// TwinCAT 3 PLC project FMStrings
// Title: FM Strings
// Company: FrameworkMonorepo
// ProjectVersion: 0.0.1
// ProgramVersion: 3.1.4024.0
// libraries:
//   FM Types, * (FrameworkMonorepo)
//   Tc2_Standard, * (Beckhoff Automation GmbH)
//   Tc2_System, * (Beckhoff Automation GmbH)
//   Tc2_Utilities, * (Beckhoff Automation GmbH)
//   Tc3_Module, * (Beckhoff Automation GmbH)
//   Base Interfaces,newest,System
// project tree:
//   Build/ BuildStringInline.TcPOU, StringBuilderExtBuffer.TcPOU, StringBuilder255.TcPOU, StringBuilderInfinite.TcPOU
//   Convert/ AnyToString.TcPOU, AnyTypeToString.TcPOU, StringToAny.TcPOU, StringToAnyType.TcPOU
//   Manipulate/ AddLeadingZeros.TcPOU, GetStringBetween.TcPOU, RemoveStringFromEnd.TcPOU, ReplaceAllAny.TcPOU, ReplaceAll.TcPOU, ReplaceAllAnyType.TcPOU, ReplaceString.TcPOU, SubString.TcPOU
//   Utf8/ Utf8String.TcDUT
//   Validate/ StringBeginsWithAny.TcPOU, StringBeginsWith.TcPOU, StringEndsWithAny.TcPOU, StringEndsWith.TcPOU
//   Version/ Global_Version.TcGVL
// (motion and I/O tree: see PLC project fmtypes)
// real-time tasks:
//   TASK BindingTestTask: cycle T#1ms, priority 20, ADS port 350
//   TASK PlcTask: cycle T#1ms, priority 21, ADS port 351
//   TASK PlcTask1: cycle T#1ms, priority 22, ADS port 352
//   TASK PlcTask2: cycle T#1ms, priority 23, ADS port 353
//   TASK MathTestTask: cycle T#1ms, priority 24, ADS port 354
//   TASK TimesTestsTask: cycle T#1ms, priority 25, ADS port 355

// ---- Utf8/Utf8String.TcDUT
{attribute 'TcEncoding':='UTF-8'}
TYPE Utf8String : T_MaxString; END_TYPE

// ---- Version/Global_Version.TcGVL
{attribute 'TcGenerated'}
{attribute 'no-analysis'}
{attribute 'linkalways'}
// This function has been automatically generated from the project information.
VAR_GLOBAL CONSTANT
	{attribute 'const_non_replaced'}
	stLibVersion_FM_Strings : ST_LibVersion := (iMajor := 0, iMinor := 0, iBuild := 1, iRevision := 0, nFlags := 0, sVersion := '0.0.1');
END_VAR

// ---- Build/BuildStringInline.TcPOU
FUNCTION BuildStringInline : REFERENCE TO StringBuilder255
VAR_INPUT
	value : T_MaxString;
END_VAR
VAR_STAT
	builder : StringBuilder255;
END_VAR

builder.Clear();

builder.Append(value);

BuildStringInline REF= builder;

END_FUNCTION

// ---- Build/StringBuilder255.TcPOU
FUNCTION_BLOCK StringBuilder255
VAR
	_Value : T_MaxString;
END_VAR

METHOD Append : REFERENCE TO StringBuilder255
VAR_INPUT
	value : T_MaxString;
END_VAR
Append REF= THIS^;

_Value := CONCAT(_Value, value);
END_METHOD

METHOD Clear : REFERENCE TO StringBuilder255
Clear REF= THIS^;

_Value := '';
END_METHOD

METHOD GetString : T_MaxString
GetString := _Value;
END_METHOD

PROPERTY IsEmpty : BOOL
GET
IsEmpty := Length = 0;
END_GET
END_PROPERTY

{attribute 'monitoring' := 'call'}
PROPERTY Length : DINT
GET
Length := LEN(_Value);
END_GET
END_PROPERTY

{attribute 'monitoring' := 'call'}
PROPERTY Value : T_MaxString
GET
Value := _Value;
END_GET
END_PROPERTY

END_FUNCTION_BLOCK

// ---- Build/StringBuilderExtBuffer.TcPOU
FUNCTION_BLOCK StringBuilderExtBuffer
VAR
	_Buffer : __SYSTEM.AnyType;
	_Length : DINT;
END_VAR

METHOD Append : REFERENCE TO StringBuilderExtBuffer
VAR_INPUT
	value : T_MaxString;
END_VAR
VAR
	lengthToCopy : DINT;
END_VAR
lengthToCopy := LIMIT(
	DINT#0, 								// min
	LEN(value), 							// value
	(_Buffer.diSize - TO_DINT(_Length) - 1) // max
);

MEMCPY(
	destAddr := _Buffer.pValue + TO_DWORD(_Length),
	srcAddr := ADR(value),
	n := TO_UDINT(lengthToCopy)
);

_Length := _Length + lengthToCopy;

Append REF= THIS^;
END_METHOD

METHOD AppendByPointer : REFERENCE TO StringBuilderExtBuffer
VAR_INPUT
	value : POINTER TO STRING;
END_VAR
VAR
	valueLength : DINT;
	lengthToCopy : DINT;
END_VAR
valueLength := TO_DINT(LEN2(value));

lengthToCopy := LIMIT(
	DINT#0, 								// min
	valueLength, 							// value
	(_Buffer.diSize - TO_DINT(_Length) - 1) // max
);

MEMCPY(
	destAddr := _Buffer.pValue + TO_DWORD(_Length),
	srcAddr := value,
	n := TO_UDINT(lengthToCopy)
);

_Length := _Length + lengthToCopy;

AppendByPointer REF= THIS^;
END_METHOD

METHOD AppendSubString : REFERENCE TO StringBuilderExtBuffer
VAR_INPUT
	value : ANY;
	startIndex : DINT;
	length : DINT;
END_VAR
VAR
	valueLength : DINT;
	lengthToCopy : DINT;
END_VAR
valueLength := length;

lengthToCopy := LIMIT(
	DINT#0, 								// min
	valueLength, 							// value
	(_Buffer.diSize - TO_DINT(_Length) - 1) // max
);

MEMCPY(
	destAddr := _Buffer.pValue + TO_DWORD(_Length),
	srcAddr := value.pValue + TO_DWORD(startIndex),
	n := TO_UDINT(lengthToCopy)
);

_Length := _Length + lengthToCopy;

AppendSubString REF= THIS^;
END_METHOD

PROPERTY Buffer : __SYSTEM.AnyType
GET
Buffer := _Buffer;
END_GET
SET
_Buffer := Buffer;
_Length := TO_DINT(LEN2(pSTRING := _Buffer.pValue));
END_SET
END_PROPERTY

{attribute 'monitoring' := 'call'}
PROPERTY BufferRef : REFERENCE TO __SYSTEM.AnyType
GET
BufferRef REF= _Buffer;
END_GET
END_PROPERTY

METHOD Clear : REFERENCE TO StringBuilderExtBuffer
MEMSET(
	destAddr := _Buffer.pValue,
	fillByte := 0,
	n := TO_UDINT(_Buffer.diSize)
);

_Length := 0;

Clear REF= THIS^;
END_METHOD

PROPERTY IsEmpty : BOOL
GET
IsEmpty := Length = 0;
END_GET
END_PROPERTY

{attribute 'monitoring' := 'call'}
PROPERTY Length : DINT
GET
Length := _Length;
END_GET
END_PROPERTY

METHOD Prepend : REFERENCE TO StringBuilderExtBuffer
VAR_INPUT
	value : T_MaxString;
END_VAR
VAR
	lengthToCopy : DINT;
END_VAR
lengthToCopy := LIMIT(
	DINT#0, 								// min
	LEN(value), 							// value
	_Buffer.diSize // max
);

MEMMOVE(
	destAddr := _Buffer.pValue + TO_DWORD(lengthToCopy),
	srcAddr := _Buffer.pValue,
	n := TO_UDINT(MIN(_Buffer.diSize - lengthToCopy, _Length))
);

MEMCPY(
	destAddr := _Buffer.pValue,
	srcAddr := ADR(value),
	n := TO_UDINT(lengthToCopy)
);

_Length := MIN(_Length + lengthToCopy, _Buffer.diSize);

Prepend REF= THIS^;
END_METHOD

METHOD UpdateBufferLength
VAR_INPUT
END_VAR
_Length := TO_DINT(LEN2(_Buffer.pValue));
END_METHOD

END_FUNCTION_BLOCK

// ---- Build/StringBuilderInfinite.TcPOU
FUNCTION_BLOCK StringBuilderInfinite
VAR
	_Capacity : DINT;
	_Length : DINT;
	_Value : POINTER TO STRING := Allocate();
END_VAR
VAR CONSTANT
	InitialCapacity : DINT := 1024;
END_VAR

METHOD PRIVATE Allocate : POINTER TO STRING
VAR
	p : POINTER TO STRING;
END_VAR
_Capacity := InitialCapacity;
p := __NEW(BYTE, TO_UDINT(_Capacity + 1));
MEMSET(destAddr := p, fillByte := 0, n := TO_UDINT(_Capacity));
Allocate := p;
END_METHOD

METHOD Append : REFERENCE TO StringBuilderInfinite
VAR_INPUT
	value : T_MaxString;
END_VAR
VAR
	lengthToCopy : DINT;
END_VAR
lengthToCopy := LEN(value);

EnsureCapacity(_Length + lengthToCopy);

MEMCPY(
	destAddr := _Value + _Length,
	srcAddr := ADR(value),
	n := TO_UDINT(lengthToCopy)
);

_Length := _Length + lengthToCopy;

Append REF= THIS^;
END_METHOD

METHOD AppendByPointer : REFERENCE TO StringBuilderInfinite
VAR_INPUT
	value : POINTER TO STRING;
END_VAR
VAR
	lengthToCopy : DINT;
END_VAR
lengthToCopy := TO_DINT(LEN2(value));

EnsureCapacity(_Length + lengthToCopy);

MEMCPY(
	destAddr := _Value + TO_LWORD(_Length),
	srcAddr := value,
	n := TO_UDINT(lengthToCopy)
);

_Length := _Length + lengthToCopy;

AppendByPointer REF= THIS^;
END_METHOD

{attribute 'monitoring' := 'call'}
PROPERTY Capacity : DINT
GET
Capacity := _Capacity;
END_GET
END_PROPERTY

METHOD Clear : REFERENCE TO StringBuilderInfinite
MEMSET(
	destAddr := _Value,
	fillByte := 0,
	n := TO_UDINT(_Length)
);

_Length := 0;

Clear REF= THIS^;
END_METHOD

METHOD PRIVATE EnsureCapacity
VAR_INPUT
	needed : DINT;
END_VAR
IF (needed < _Capacity) THEN
	RETURN;
END_IF

IF (needed > _Capacity * 2) THEN
	_Capacity := needed;
ELSE
	_Capacity := NextPowerOf2(needed);
END_IF

Reallocate();
END_METHOD

METHOD FB_exit : BOOL
VAR_INPUT
	bInCopyCode : BOOL; // if TRUE, the exit method is called for exiting an instance that is copied afterwards (online change).
END_VAR
__DELETE(_Value);
END_METHOD

PROPERTY IsEmpty : BOOL
GET
IsEmpty := Length = 0;
END_GET
END_PROPERTY

{attribute 'monitoring' := 'call'}
PROPERTY Length : DINT
GET
Length := _Length;
END_GET
END_PROPERTY

METHOD PRIVATE NextPowerOf2 : DINT
VAR_INPUT
	number : DINT;
END_VAR
VAR
	n : UDINT;
END_VAR
n := TO_UDINT(number);
n := n - 1;
n := n OR SHR(n, 1);
n := n OR SHR(n, 2);
n := n OR SHR(n, 4);
n := n OR SHR(n, 8);
n := n OR SHR(n, 16);
n := n + 1;
NextPowerOf2 := TO_DINT(n);
END_METHOD

METHOD PRIVATE Reallocate
VAR_INPUT
END_VAR
VAR
	new : POINTER TO STRING;
END_VAR
new := __NEW(BYTE, TO_UDINT(_Capacity + 1));
MEMSET(destAddr := new, fillByte := 0, n := TO_UDINT(_Capacity));
MEMCPY(new, _Value, TO_UDINT(_Length));
__DELETE(_Value);
_Value := new;
END_METHOD

{attribute 'monitoring' := 'call'}
PROPERTY Value : POINTER TO STRING(1000)
GET
Value := _Value;
END_GET
END_PROPERTY

END_FUNCTION_BLOCK

// ---- Convert/AnyToString.TcPOU
FUNCTION AnyToString : T_MaxString
VAR_INPUT
	a : ANY;
END_VAR

AnyToString := AnyTypeToString(a);

END_FUNCTION

// ---- Convert/AnyTypeToString.TcPOU
FUNCTION AnyTypeToString : T_MaxString
VAR_INPUT
	a : __SYSTEM.AnyType;
END_VAR

CASE UDINT_TO_INT(a.TypeClass) OF
    IBaseLibrary.TypeClass.TYPE_BOOL :
        AnyTypeToString := BOOL_TO_STRING(PBOOL_TO_BOOL(a.pValue));
    IBaseLibrary.TypeClass.TYPE_BYTE :
        AnyTypeToString := BYTE_TO_STRING(a.pValue^);
    IBaseLibrary.TypeClass.TYPE_WORD :
        AnyTypeToString := WORD_TO_STRING(PWORD_TO_WORD(a.pValue));
    IBaseLibrary.TypeClass.TYPE_DWORD :
        AnyTypeToString := DWORD_TO_STRING(PDWORD_TO_DWORD(a.pValue));
    IBaseLibrary.TypeClass.TYPE_LWORD :
        AnyTypeToString := LWORD_TO_STRING(PLWORD_TO_LWORD(a.pValue));
    IBaseLibrary.TypeClass.TYPE_SINT :
        AnyTypeToString := SINT_TO_STRING(PSINT_TO_SINT(a.pValue));
    IBaseLibrary.TypeClass.TYPE_INT :
        AnyTypeToString := INT_TO_STRING(PINT_TO_INT(a.pValue));
    IBaseLibrary.TypeClass.TYPE_DINT :
        AnyTypeToString := DINT_TO_STRING(PDINT_TO_DINT(a.pValue));
    IBaseLibrary.TypeClass.TYPE_LINT :
        AnyTypeToString := LINT_TO_STRING(PLINT_TO_LINT(a.pValue));
    IBaseLibrary.TypeClass.TYPE_USINT :
        AnyTypeToString := USINT_TO_STRING(PUSINT_TO_USINT(a.pValue));
    IBaseLibrary.TypeClass.TYPE_UINT :
        AnyTypeToString := UINT_TO_STRING(PUINT_TO_UINT(a.pValue));
    IBaseLibrary.TypeClass.TYPE_UDINT :
        AnyTypeToString := UDINT_TO_STRING(PUDINT_TO_UDINT(a.pValue));
    IBaseLibrary.TypeClass.TYPE_ULINT :
        AnyTypeToString := ULINT_TO_STRING(PULINT_TO_ULINT(a.pValue));
    IBaseLibrary.TypeClass.TYPE_REAL :
        AnyTypeToString := REAL_TO_STRING(PREAL_TO_REAL(a.pValue));
    IBaseLibrary.TypeClass.TYPE_LREAL :
        AnyTypeToString := LREAL_TO_STRING(PLREAL_TO_LREAL(a.pValue));
    IBaseLibrary.TypeClass.TYPE_STRING :
		AnyTypeToString := PMAXSTRING_TO_MAXSTRING(a.pValue);
    IBaseLibrary.TypeClass.TYPE_TIME :
        AnyTypeToString := TIME_TO_STRING(PTIME_TO_TIME(a.pValue));
    IBaseLibrary.TypeClass.TYPE_DATE :
        AnyTypeToString := DATE_TO_STRING(PDATE_TO_DATE(a.pValue));
    IBaseLibrary.TypeClass.TYPE_DATEANDTIME :
        AnyTypeToString := DT_TO_STRING(PDT_TO_DT(a.pValue));
    IBaseLibrary.TypeClass.TYPE_TIMEOFDAY :
        AnyTypeToString := TOD_TO_STRING(PTOD_TO_TOD(a.pValue));
    IBaseLibrary.TypeClass.TYPE_POINTER :
        AnyTypeToString := PVOID_TO_HEXSTR(a.pValue, SIZEOF(PVOID), FALSE);
    IBaseLibrary.TypeClass.TYPE_LTIME :
        AnyTypeToString := LTIME_TO_STRING(PLTIME_TO_LTIME(a.pValue));
    ELSE
        AnyTypeToString := 'ERROR: UNSUPPORTED DATA TYPE';
END_CASE

END_FUNCTION

// ---- Convert/StringToAny.TcPOU
FUNCTION StringToAny
VAR_INPUT
	text : T_MaxString;
	output : ANY;
END_VAR

StringToAnyType(text, output);

END_FUNCTION

// ---- Convert/StringToAnyType.TcPOU
FUNCTION StringToAnyType
VAR_INPUT
	text : T_MaxString;
	output : __SYSTEM.AnyType;
END_VAR
VAR
	conversion : AnyTypeUnion;
END_VAR

CASE UDINT_TO_INT(output.TypeClass) OF
    IBaseLibrary.TypeClass.TYPE_BOOL :
        conversion.BOOL_ := STRING_TO_BOOL(text);
        MEMCPY(srcAddr := ADR(conversion.BOOL_), destAddr := output.pValue, n := TO_UDINT(MIN(output.diSize, SIZEOF(conversion.BOOL_))));
    IBaseLibrary.TypeClass.TYPE_BYTE :
        conversion.BYTE_ := STRING_TO_BYTE(text);
        MEMCPY(srcAddr := ADR(conversion.BYTE_), destAddr := output.pValue, n := TO_UDINT(MIN(output.diSize, SIZEOF(conversion.BYTE_))));
    IBaseLibrary.TypeClass.TYPE_WORD :
        conversion.WORD_ := STRING_TO_WORD(text);
        MEMCPY(srcAddr := ADR(conversion.WORD_), destAddr := output.pValue, n := TO_UDINT(MIN(output.diSize, SIZEOF(conversion.WORD_))));
    IBaseLibrary.TypeClass.TYPE_DWORD :
        conversion.DWORD_ := STRING_TO_DWORD(text);
        MEMCPY(srcAddr := ADR(conversion.DWORD_), destAddr := output.pValue, n := TO_UDINT(MIN(output.diSize, SIZEOF(conversion.DWORD_))));
    IBaseLibrary.TypeClass.TYPE_LWORD :
        conversion.LWORD_ := STRING_TO_LWORD(text);
        MEMCPY(srcAddr := ADR(conversion.LWORD_), destAddr := output.pValue, n := TO_UDINT(MIN(output.diSize, SIZEOF(conversion.LWORD_))));
    IBaseLibrary.TypeClass.TYPE_SINT :
        conversion.SINT_ := STRING_TO_SINT(text);
        MEMCPY(srcAddr := ADR(conversion.SINT_), destAddr := output.pValue, n := TO_UDINT(MIN(output.diSize, SIZEOF(conversion.SINT_))));
    IBaseLibrary.TypeClass.TYPE_INT :
        conversion.INT_ := STRING_TO_INT(text);
        MEMCPY(srcAddr := ADR(conversion.INT_), destAddr := output.pValue, n := TO_UDINT(MIN(output.diSize, SIZEOF(conversion.INT_))));
    IBaseLibrary.TypeClass.TYPE_DINT :
        conversion.DINT_ := STRING_TO_DINT(text);
        MEMCPY(srcAddr := ADR(conversion.DINT_), destAddr := output.pValue, n := TO_UDINT(MIN(output.diSize, SIZEOF(conversion.DINT_))));
    IBaseLibrary.TypeClass.TYPE_LINT :
        conversion.LINT_ := STRING_TO_LINT(text);
        MEMCPY(srcAddr := ADR(conversion.LINT_), destAddr := output.pValue, n := TO_UDINT(MIN(output.diSize, SIZEOF(conversion.LINT_))));
    IBaseLibrary.TypeClass.TYPE_USINT :
        conversion.USINT_ := STRING_TO_USINT(text);
        MEMCPY(srcAddr := ADR(conversion.USINT_), destAddr := output.pValue, n := TO_UDINT(MIN(output.diSize, SIZEOF(conversion.USINT_))));
    IBaseLibrary.TypeClass.TYPE_UINT :
        conversion.UINT_ := STRING_TO_UINT(text);
        MEMCPY(srcAddr := ADR(conversion.UINT_), destAddr := output.pValue, n := TO_UDINT(MIN(output.diSize, SIZEOF(conversion.UINT_))));
    IBaseLibrary.TypeClass.TYPE_UDINT :
        conversion.UDINT_ := STRING_TO_UDINT(text);
        MEMCPY(srcAddr := ADR(conversion.UDINT_), destAddr := output.pValue, n := TO_UDINT(MIN(output.diSize, SIZEOF(conversion.UDINT_))));
    IBaseLibrary.TypeClass.TYPE_ULINT :
        conversion.ULINT_ := STRING_TO_ULINT(text);
        MEMCPY(srcAddr := ADR(conversion.ULINT_), destAddr := output.pValue, n := TO_UDINT(MIN(output.diSize, SIZEOF(conversion.ULINT_))));
    IBaseLibrary.TypeClass.TYPE_REAL :
        conversion.REAL_ := STRING_TO_REAL(text);
        MEMCPY(srcAddr := ADR(conversion.REAL_), destAddr := output.pValue, n := TO_UDINT(MIN(output.diSize, SIZEOF(conversion.REAL_))));
    IBaseLibrary.TypeClass.TYPE_LREAL :
        conversion.LREAL_ := STRING_TO_LREAL(text);
        MEMCPY(srcAddr := ADR(conversion.LREAL_), destAddr := output.pValue, n := TO_UDINT(MIN(output.diSize, SIZEOF(conversion.LREAL_))));
    IBaseLibrary.TypeClass.TYPE_STRING :
        conversion.STRING_ := text;
        MEMCPY(srcAddr := ADR(conversion.STRING_), destAddr := output.pValue, n := TO_UDINT(MIN(output.diSize, SIZEOF(conversion.STRING_))));
    IBaseLibrary.TypeClass.TYPE_TIME :
        conversion.TIME_ := STRING_TO_TIME(text);
        MEMCPY(srcAddr := ADR(conversion.TIME_), destAddr := output.pValue, n := TO_UDINT(MIN(output.diSize, SIZEOF(conversion.TIME_))));
    IBaseLibrary.TypeClass.TYPE_DATE :
        conversion.DATE_ := STRING_TO_DATE(text);
        MEMCPY(srcAddr := ADR(conversion.DATE_), destAddr := output.pValue, n := TO_UDINT(MIN(output.diSize, SIZEOF(conversion.DATE_))));
    IBaseLibrary.TypeClass.TYPE_DATEANDTIME :
        conversion.DATEANDTIME_ := STRING_TO_DT(text);
        MEMCPY(srcAddr := ADR(conversion.DATEANDTIME_), destAddr := output.pValue, n := TO_UDINT(MIN(output.diSize, SIZEOF(conversion.DATEANDTIME_))));
    IBaseLibrary.TypeClass.TYPE_TIMEOFDAY :
        conversion.TIMEOFDAY_ := STRING_TO_TOD(text);
        MEMCPY(srcAddr := ADR(conversion.TIMEOFDAY_), destAddr := output.pValue, n := TO_UDINT(MIN(output.diSize, SIZEOF(conversion.TIMEOFDAY_))));
    IBaseLibrary.TypeClass.TYPE_POINTER :
        conversion.POINTER_ := STRING_TO_PVOID(text);
        MEMCPY(srcAddr := ADR(conversion.POINTER_), destAddr := output.pValue, n := TO_UDINT(MIN(output.diSize, SIZEOF(conversion.POINTER_))));
    IBaseLibrary.TypeClass.TYPE_LTIME :
        conversion.LTIME_ := STRING_TO_LTIME(text);
        MEMCPY(srcAddr := ADR(conversion.LTIME_), destAddr := output.pValue, n := TO_UDINT(MIN(output.diSize, SIZEOF(conversion.LTIME_))));
END_CASE

END_FUNCTION

// ---- Manipulate/AddLeadingZeros.TcPOU
FUNCTION AddLeadingZeros : STRING
VAR_INPUT
	str : STRING;
	charNumber : USINT;
END_VAR

AddLeadingZeros := str;
IF charNumber > LEN(str) THEN
	AddLeadingZeros := CONCAT('0', AddLeadingZeros);
	AddLeadingZeros := .AddLeadingZeros(AddLeadingZeros, charNumber);
END_IF

END_FUNCTION

// ---- Manipulate/GetStringBetween.TcPOU
FUNCTION GetStringBetween : T_MaxString
VAR_INPUT
	searched : T_MaxString;
	left : T_MaxString;
	right : T_MaxString;
END_VAR
VAR
	leftIndex : INT;
	rightIndex : INT;
	offset : INT;
END_VAR

leftIndex := FIND(searched, left);
IF (leftIndex = 0) THEN
	RETURN;
END_IF
offset := leftIndex + LEN(left);
rightIndex := TO_INT(FIND2(ADR(searched[offset]) - 1, ADR(right)));
IF (rightIndex = 0) THEN
	RETURN;
END_IF
GetStringBetween := 
	MID(STR := searched, POS := offset, LEN := rightIndex - 1);

END_FUNCTION

// ---- Manipulate/RemoveStringFromEnd.TcPOU
FUNCTION RemoveStringFromEnd : T_MaxString
VAR_INPUT
	text : T_MaxString;
	end : T_MaxString;
END_VAR
VAR
	diff : INT;
END_VAR

diff := LEN(text) - LEN(end);
IF (diff < 0) THEN
	RemoveStringFromEnd := text;
	RETURN;
END_IF

IF (StringEndsWithAny(text, end)) THEN
	RemoveStringFromEnd := LEFT(text, diff);
END_IF

END_FUNCTION

// ---- Validate/StringEndsWithAny.TcPOU
FUNCTION StringEndsWithAny : BOOL
VAR_INPUT
	text : ANY;
	endsWithString : T_MaxString;
END_VAR
VAR
	textLength : DINT;
	length : DINT;
END_VAR

textLength := TO_DINT(LEN2(text.pValue));
length := LEN(endsWithString);

IF (textLength < length) THEN
	RETURN;
END_IF

StringEndsWithAny := MEMCMP(pBuf1 := text.pValue + TO_DWORD(textLength - length), pBuf2 := ADR(endsWithString), n := TO_UDINT(length)) = 0;

END_FUNCTION

// ---- Manipulate/ReplaceAllAny.TcPOU
FUNCTION ReplaceAllAny
VAR_INPUT
	in : ANY;
	replaced : T_MaxString;
	with : T_MaxString;
END_VAR

ReplaceAllAnyType(in, replaced, with);

END_FUNCTION

// ---- Manipulate/ReplaceAllAnyType.TcPOU
FUNCTION ReplaceAllAnyType
VAR_INPUT
	in : __SYSTEM.AnyType;
	replaced : T_MaxString;
	with : T_MaxString;
END_VAR
VAR
	new : POINTER TO BYTE;
END_VAR

IF (FIND2(in.pValue, ADR(replaced)) = 0) THEN
	RETURN;
END_IF

new := __NEW(BYTE, TO_UDINT(in.diSize));

FindAndReplace(
	pSrcString := in.pValue,
	pDeleteString := ADR(replaced),
	pInsertString := ADR(with),
	pDstString := new,
	nDstSize := TO_UDINT(in.diSize - 1)
);

MEMCPY(in.pValue, new, TO_UDINT(in.diSize));
__DELETE(new);

END_FUNCTION

// ---- Manipulate/ReplaceAll.TcPOU
FUNCTION ReplaceAll : T_MaxString
VAR_INPUT
	in : T_MaxString;
	replaced : T_MaxString;
	with : T_MaxString;
END_VAR

IF (FIND(in, replaced) = 0) THEN
	ReplaceAll := in;
	RETURN;
END_IF

FindAndReplace(
	pSrcString := ADR(in),
	pDeleteString := ADR(replaced),
	pInsertString := ADR(with),
	pDstString := ADR(ReplaceAll),
	nDstSize := SIZEOF(ReplaceAll) - 1
);

END_FUNCTION

// ---- Manipulate/ReplaceString.TcPOU
FUNCTION ReplaceString
VAR_INPUT
	in : ANY;
	replaced : T_MaxString;
	with : T_MaxString;
END_VAR
VAR
	replaceBegin : UDINT;
END_VAR

replaceBegin := FIND2(in.pValue, ADR(replaced));

IF (replaceBegin = 0) THEN
	RETURN;
END_IF

REPLACE2(in.pValue, ADR(with), in.pValue, TO_UDINT(in.diSize), TO_UDINT(LEN(replaced)), replaceBegin);

END_FUNCTION

// ---- Manipulate/SubString.TcPOU
FUNCTION SubString
VAR_INPUT
	source : ANY;
	destination : ANY;
	startIndex : DINT;
	length : DINT;
END_VAR
VAR
END_VAR

IF (startIndex >= source.diSize) THEN
	RETURN;
END_IF

MEMCPY(
	destAddr := destination.pValue,
	srcAddr := source.pValue + TO_DWORD(startIndex),
	n := TO_UDINT(MIN(length, MIN(source.diSize - startIndex, destination.diSize)))
);

END_FUNCTION

// ---- Validate/StringBeginsWithAny.TcPOU
FUNCTION StringBeginsWithAny : BOOL
VAR_INPUT
	text : ANY;
	startsWithString : T_MaxString;
END_VAR
VAR
	textLength : DINT;
	length : DINT;
END_VAR

textLength := TO_DINT(LEN2(text.pValue));
length := LEN(startsWithString);

IF (textLength < length) THEN
	RETURN;
END_IF

StringBeginsWithAny := MEMCMP(pBuf1 := text.pValue, pBuf2 := ADR(startsWithString), n := TO_UDINT(length)) = 0;

END_FUNCTION

// ---- Validate/StringBeginsWith.TcPOU
FUNCTION StringBeginsWith : BOOL
VAR_INPUT
	text : T_MaxString;
	startsWithString : T_MaxString;
END_VAR
VAR
	textLength : DINT;
	length : DINT;
END_VAR

textLength := LEN(text);
length := LEN(startsWithString);

IF (textLength < length) THEN
	RETURN;
END_IF

StringBeginsWith := MEMCMP(pBuf1 := ADR(text), pBuf2 := ADR(startsWithString), n := TO_UDINT(length)) = 0;

END_FUNCTION

// ---- Validate/StringEndsWith.TcPOU
FUNCTION StringEndsWith : BOOL
VAR_INPUT
	text : T_MaxString;
	endsWithString : T_MaxString;
END_VAR
VAR
	textLength : DINT;
	length : DINT;
END_VAR

textLength := LEN(text);
length := LEN(endsWithString);

IF (textLength < length) THEN
	RETURN;
END_IF

StringEndsWith := MEMCMP(pBuf1 := ADR(text) + TO_DWORD(textLength - length), pBuf2 := ADR(endsWithString), n := TO_UDINT(length)) = 0;

END_FUNCTION
